// TwinCAT 3 PLC project MyPLC
// ProgramVersion: 3.1.4023.0
// libraries:
//   Tc2_Standard, * (Beckhoff Automation GmbH)
//   Tc2_System, * (Beckhoff Automation GmbH)
//   Tc3_Module, * (Beckhoff Automation GmbH)
// project tree:
//   DUTs/ E_Options.TcDUT, MyStructure.TcDUT, MyStructureExtended.TcDUT
//   GVLs/ GVL_Main.TcGVL
//   / PlcTask.TcTTO
//   POUs/ FB_MyBlock.TcPOU, FB_SecondBlock.TcPOU, MAIN.TcPOU, PlainFunction.TcPOU, PlainFunctionBlock.TcPOU, RegularFunction.TcPOU
// real-time tasks:
//   TASK PlcTask: cycle T#10ms, priority 20, ADS port 350

CONFIGURATION MyPLC
    RESOURCE PLC ON TwinCAT3
        TASK PlcTask(INTERVAL := T#10ms, PRIORITY := 20);
        PROGRAM MAIN WITH PlcTask : MAIN;
    END_RESOURCE
END_CONFIGURATION

// ---- DUTs/E_Options.TcDUT
{attribute 'qualified_only'}
{attribute 'strict'}
TYPE E_Options :
(
	Default := 0,
    Option1,
    Option2
);
END_TYPE

// ---- DUTs/MyStructure.TcDUT
TYPE MyStructure :
STRUCT
    member1     : LREAL; // Some member
END_STRUCT
END_TYPE

// ---- DUTs/MyStructureExtended.TcDUT
TYPE MyStructureExtended EXTENDS MyStructure :
STRUCT
    member2     : UDINT;            //          Another property
END_STRUCT
END_TYPE

// ---- GVLs/GVL_Main.TcGVL
{attribute 'qualified_only'}
(*
Some global variable list.

Access must include the file name!
*)
VAR_GLOBAL
    someGlobal      : LREAL;    // Description 1
    otherGlobal     : INT;      // Description 2
END_VAR

// ---- POUs/MAIN.TcPOU
PROGRAM MAIN
VAR
    request         : UDINT := 0;
    ack             : UDINT := 0;
    
    block           : FB_MyBlock;
    
    result          : LREAL;
    
END_VAR

IF ack <> request THEN
    ack := request;
END_IF

result := RegularFunction(input := 3.14, other_arg := 7);

END_PROGRAM

// ---- POUs/FB_MyBlock.TcPOU
(*
Info!
*)
FUNCTION_BLOCK FB_MyBlock
VAR_INPUT
    someInput       : LREAL;        // This is some input with a description
    otherInput      : BOOL;         // Awesome description 
END_VAR
VAR_INPUT
    secondClause    : LREAL;        // This is some input with a description 
END_VAR
VAR_OUTPUT
    myOutput        : UINT;         // Return something nice
END_VAR
VAR
END_VAR

myOutput := 420;

METHOD AnotherMethod : LREAL
VAR_INPUT
    methodInput     : LREAL;            // Some input
END_VAR
END_METHOD

(*
This is a description.
*)
METHOD MyMethod : BOOL
VAR_INPUT
END_VAR
MyMethod := FALSE;
END_METHOD

END_FUNCTION_BLOCK

// ---- POUs/RegularFunction.TcPOU
(*
Short description of the function.

Long description of the function, spanning multiple
rows even.
*)
FUNCTION RegularFunction : LREAL
VAR_INPUT
    input       : LREAL;            // This is an in-code description of some variable
    other_arg   : UDINT;
END_VAR
VAR
END_VAR

RegularFunction := input * 2.0;

END_FUNCTION

// ---- POUs/FB_SecondBlock.TcPOU
FUNCTION_BLOCK FB_SecondBlock EXTENDS FB_MyBlock
VAR_INPUT
END_VAR
VAR_OUTPUT
END_VAR
VAR
END_VAR

END_FUNCTION_BLOCK

// ---- POUs/PlainFunction.TcPOU
FUNCTION PlainFunction : BOOL
VAR_INPUT
END_VAR
VAR
END_VAR

END_FUNCTION

// ---- POUs/PlainFunctionBlock.TcPOU
FUNCTION_BLOCK PlainFunctionBlock
VAR_INPUT
    someInput       : BOOL;
END_VAR
VAR_OUTPUT
    someOutput      : BOOL;
END_VAR
VAR
END_VAR

END_FUNCTION_BLOCK
